FUNCTION_BLOCK FB_TEST_CheckPartCapperFail EXTENDS FB_Test
VAR
END_VAR

METHOD Execute : ST_TestResults
VAR
	MockStatus		: ST_PartStatus;
	fbCell			: FB_Cell;
	testExpected	: BOOL;
	testResult		: BOOL;
END_VAR
MockStatus.bBarcodeStatus := TRUE;
MockStatus.bCapperStatus := FALSE;
MockStatus.bFillerStatus := TRUE;
MockStatus.bWeightStatus := TRUE;

testExpected := FALSE;
testResult := fbCell.CheckPart(MockStatus);

Execute := AssertEquals(
	testExpected, 
	testResult, 
	'Part status fail.'
);
END_METHOD

END_FUNCTION_BLOCK

(* stored: Version 1.1.0.1, ProductVersion 3.1.4024.12
   POU FB_TEST_CheckPartCapperFail: Id {2c821e1b-9a43-4664-ad77-e4e71fe3d5a1}, SpecialFunc None
   Method Execute: Id {6e443ba0-a0ea-4732-bae1-232a01610c9c} *)
